# B&R Automation Studio project TD52 (part 28)

#### Ctr_CCCyclic.st
```iecst
(*******************************************************************************
Ctr_CC

This code is confidential and proprietary to the INNIO Company.
It may not be used in any form, or reproduced in any manner,
without the express written permission of the INNIO Company.
Copyright, INNIO Company, 2022

Customized modifications: -
------------------------

History:
-------
V4.x.x		14.01.2015	Walid Mari  	copied from Ctr_ECW
V4.00.1		25.06.2015	lettenbichler	twice declared par.removed
V4.11.0		28.01.2022	Perktold		included plant controller upgrade

Instructions for use:
--------------------

Outstandings:
------------
(*******************************************************************************)

PROGRAM _CYCLIC

	(* Parameter *)
	Para.tCtr_CC.W_set;
	Para.tCtr_CC.W_set2;
	Para.tCtr_CC.W_min;
	Para.tCtr_CC.W_max;
	Para.tCtr_CC.dW_up;
	Para.tCtr_CC.dW_down;
	Para.tCtr_CC.deadband;
	Para.tCtr_CC.Y_min;
	Para.tCtr_CC.Y_max;
	Para.tCtr_CC.dY_max;
	Para.tCtr_CC.Y_block;
	Para.tCtr_CC.invert;
	Para.tCtr_CC.Kp;
	Para.tCtr_CC.Tn;
	Para.tCtr_CC.Tv;
	Para.tCtr_CC.Kp_GainScheduling;
	Para.tCtr_CC.Tn_GainScheduling;
	Para.tCtr_CC.Tv_GainScheduling;

	(* Input variables *)
	tCtr_CC_In	 				:= VIS2MM.tCtr_CC_In;			(* from vis *)

	(* Input from module *)
	tCtr_CC_In.enable			:= OUT_AG.tBbBlower.Do		AND
								   Para.bCtr_CC 			AND
								   Para.bPr_CC_MS_Exist		AND
								   IN_AG.tPB2MM.bParaSetupOk;

	tCtr_CC_In.W_ext_Active		:= tCtr_CC_In.W_ext_Active;		(* from vis *)
	tCtr_CC_In.W_ext			:= 0.0;
	tCtr_CC_In.Y_set_Active		:= FALSE;
	tCtr_CC_In.Y_set			:= 0.0;
	tCtr_CC_In.X				:= IN_AG.tPr_CC.Ai;
	tCtr_CC_In.A				:= 0;
	tCtr_CC_In.W_set2_Active	:= FALSE;	(*Input to define which internal setpoint will be used TRUE = use the 2nd set point | FALSE use the normal "1st" one*)
	tCtr_CC_In.GainScheduling	:= 0.0;		(*Input for Gain Scheduling: 0.0 = use 100% of the Standard PID-Parameters | 1.0 = use 100% of the GainSched. PID Parameters | linear interpolation in between*)
	tCtr_CC_In.Y_min_cust		:= -1.0;	(*"customized" Y-Min at the current moment (The existing Y-Min parameter is the global minimum. To have an effect Y_min_cust needs to be > the parameter | -1.0 = function not used*)
	tCtr_CC_In.Y_max_cust		:= 1.0;		(*"customized" Y-Max at the current moment (The existing Y-Max parameter is the global maximum. To have an effect Y_max_cust needs to be < the parameter | 1.0 = function not used*)
	tCtr_CC_In.Retrigger		:= FALSE;	(*a rising edge on this input signals the controller to retrigger - set W on X and force the Integrator to the current Y*)

	(* Input from Visualization via OPC *)
	tCtr_CC_In.Y_man_Active;
	tCtr_CC_In.Y_man;
	tCtr_CC_In.X_min;
	tCtr_CC_In.X_max;
	tCtr_CC_In.Tune_quality;
	tCtr_CC_In.Tune_PI;
	tCtr_CC_In.Tune_PID;
	tCtr_CC_In.Tune_start;
	tCtr_CC_In.Tune_stop;
	tCtr_CC_In.Tune_takeover;

	xCtr_CC();

	(* Output variables function block *)
	(* Output to module(s) *)
	rPc_BbBlower 				:= tCtr_CC_Out.Y;	(* analog out *)

	(* Output to Visualization via OPC *)
	MM2VIS.tCtr_CC_Out			:= tCtr_CC_Out;
	VIS2MM.tCtr_CC_In			:= tCtr_CC_In;		(* write back to IN_struct for reset: Tune_takeover, X-display, ...!*)

	tCtr_CC_Out.Active;
	tCtr_CC_Out.Y;
	tCtr_CC_Out.W;
	tCtr_CC_Out.e;
	tCtr_CC_Out.Kp_tune;
	tCtr_CC_Out.Tn_tune;
	tCtr_CC_Out.Tv_tune;
	tCtr_CC_Out.status;

END_PROGRAM
```

#### Ctr_CCInit.st
```iecst
PROGRAM _INIT

	xCtr_CC.pParameter 	:= ADR(Para.tCtr_CC);
	xCtr_CC.pInput 	 	:= ADR(tCtr_CC_In);
	xCtr_CC.pOutput	 	:= ADR(tCtr_CC_Out);

	tCtr_CC_In.AlwaysUseYRamp		:= TRUE;	(*If TRUE the Y signal will always limit the change rate via the according parameter | if FALSE the Y signal will jump in case the controller is disabled (blocked or set)*)
	tCtr_CC_In.KeepYManAtBlock		:= TRUE;	(*If TRUE the controller will keep the Y-man value constant in case the controller is disabled (blocked or set) | If FALSE the blocked or set value will override the Y-man value*)
	tCtr_CC_In.Y_min_cust			:= -1.0;	(*"customized" Y-Min at the current moment (The existing Y-Min parameter is the global minimum. To have an effect Y_min_cust needs to be > the parameter | -1.0 = function not used*)
	tCtr_CC_In.Y_max_cust			:=  1.0;	(*"customized" Y-Max at the current moment (The existing Y-Max parameter is the global maximum. To have an effect Y_max_cust needs to be < the parameter | 1.0 = function not used*)
	tCtr_CC_In.StepperMode			:= FALSE;	(* TRUE = use PWM-Mode (standard mode until 4.10) | FALSE = use continuous servo drive *)
END_PROGRAM
```

### Program Logical/AuxiliariesGeneral/Ctr_ECW (IEC, version 4.12.0) - controller engine cooling water

#### Ctr_ECWCyclic.st
```iecst
(*******************************************************************************
Ctr_ECW		controller engine cooling water temperature

This code is confidential and proprietary to the INNIO Company.
It may not be used in any form, or reproduced in any manner,
without the express written permission of the INNIO Company.
Copyright, INNIO Company, 2022

Customized modifications: -
------------------------

History:
-------
V3.90.0		01.10.2012	lettenb.	new for series 9
			23.11.2012	lettenb.	write back to IN_struct added (zengerer)
V4.00.0		15.12.2014				work around(920 stapelfeld)
V4.03.0     11.01.2016              temporarily para set after controller start added
V4.03.1		03.10.2016  Fahringer	modified controller and ramp start(GeACtr with AntiWindUp)
									canceled 3 min. Tv after controller start
V4.04.0		23.03.2017	lettenb.	init restored for GeACtr with AntiWindUp
V4.05.0 	20.09.2017	Messner		Active Cooling Program added
V4.07.0		04.04.2019	Fahringer	restart the controller to initiate the setpoint ramp
			20.05.2019	Schmid		bCtrDisable was missing in tCtr_ECW_In.enable
V4.11.0		28.01.2022	Perktold	included plant controller upgrade
V4.12.0		14.12.2022	Perktold	retrigger caused by X >= WMin just once per controller activation

Instructions for use:
--------------------

Outstandings:
------------
(*******************************************************************************)

PROGRAM _CYCLIC

	(* Parameter *)
	Para.tCtr_ECW.W_set;
	Para.tCtr_ECW.W_set2;
	Para.tCtr_ECW.W_min;
	Para.tCtr_ECW.W_max;
	Para.tCtr_ECW.dW_up;
	Para.tCtr_ECW.dW_down;
	Para.tCtr_ECW.deadband;
	Para.tCtr_ECW.Y_min;
	Para.tCtr_ECW.Y_max;
	Para.tCtr_ECW.dY_max;
	Para.tCtr_ECW.Y_block;
	Para.tCtr_ECW.invert;
	Para.tCtr_ECW.Kp;
	Para.tCtr_ECW.Tn;
	Para.tCtr_ECW.Tv;
	Para.tCtr_ECW.Kp_GainScheduling;
	Para.tCtr_ECW.Tn_GainScheduling;
	Para.tCtr_ECW.Tv_GainScheduling;
	Para.tCtr_ECW.t_min_pulse_down;
	Para.tCtr_ECW.t_min_pulse_up;
	Para.tCtr_ECW.t_period_down;
	Para.tCtr_ECW.t_period_up;

	(* Input variables *)
	tCtr_ECW_In	 				:= VIS2MM.tCtr_ECW_In;			(* from vis *)

	(* Input from module *)
	tCtr_ECW_In.enable			:=	IN_AG.tPB2MM.bParaSetupOk
								AND	Para.bCtr_ECW
								AND IN_AG.bEng_Aux_Dem_CDR
								AND bCtr_ECW_Activation;

	(* start controller when actual value X reached the minimum setpoint W_min *)
	IF tCtr_ECW_In.X >= Para.tCtr_ECW.W_min THEN
		bCtr_ECW_Activation := TRUE;
	ELSE
		bCtr_ECW_Activation := tCtr_ECW_In.enable;
	END_IF;

	(* Active Cooling Program - valve setpoint *)
	IF IN_AG.bEng_Aux_Dem_CDR THEN
		tCtr_ECW_In.Y_set_Active	:= FALSE;
		tCtr_ECW_In.Y_set			:= 0.0;
	ELSE
		tCtr_ECW_In.Y_set_Active	:= bACP_Start AND NOT bACP_ECW_Cmp AND OUT_AG.tECWP1Dem.Do;
		tCtr_ECW_In.Y_set			:= 1.0;
	END_IF;

	tCtr_ECW_In.W_ext_Active	:= tCtr_ECW_In.W_ext_Active;	(* from vis *)
	tCtr_ECW_In.W_ext			:= 0.0;
	tCtr_ECW_In.X				:= IN_AG.tT_ECW.Ai;
	tCtr_ECW_In.A				:= 0;
	tCtr_ECW_In.W_set2_Active	:= FALSE;	(*Input to define which internal setpoint will be used TRUE = use the 2nd set point | FALSE use the normal "1st" one*)
	tCtr_ECW_In.GainScheduling	:= 0.0;		(*Input for Gain Scheduling: 0.0 = use 100% of the Standard PID-Parameters | 1.0 = use 100% of the GainSched. PID Parameters | linear interpolation in between*)
	tCtr_ECW_In.Y_min_cust		:= -1.0;	(*"customized" Y-Min at the current moment (The existing Y-Min parameter is the global minimum. To have an effect Y_min_cust needs to be > the parameter | -1.0 = function not used*)
	tCtr_ECW_In.Y_max_cust		:= 1.0;		(*"customized" Y-Max at the current moment (The existing Y-Max parameter is the global maximum. To have an effect Y_max_cust needs to be < the parameter | 1.0 = function not used*)

	(* retrigger controller when Ctrl.X reached the minimum set point W_min and GCB is closed  OR closure of GCB*)
	tCtr_ECW_In.Retrigger	:= (EDGEPOS(tCtr_ECW_In.X >= Para.tCtr_ECW.W_min) AND NOT bBlockRetrigger) OR EDGEPOS(IN_AG.tGCB_On.Di);

	(* block retrigger caused be X >= WMin after one execution until controller is disabled again *)
	IF tCtr_ECW_In.Retrigger AND EDGEPOS(tCtr_ECW_In.X >= Para.tCtr_ECW.W_min) THEN
		bBlockRetrigger	:= TRUE;
	ELSIF bBlockRetrigger AND NOT tCtr_ECW_In.enable THEN
		bBlockRetrigger	:= FALSE;
	END_IF;

	(* Input from Visualization via OPC *)
	tCtr_ECW_In.Y_man_Active;
	tCtr_ECW_In.Y_man;
	tCtr_ECW_In.X_min;
	tCtr_ECW_In.X_max;
	tCtr_ECW_In.Tune_quality;
	tCtr_ECW_In.Tune_PI;
	tCtr_ECW_In.Tune_PID;
	tCtr_ECW_In.Tune_start;
	tCtr_ECW_In.Tune_stop;
	tCtr_ECW_In.Tune_takeover;

	xCtr_ECW();

	(* Output variables function block *)
	(* Output to module(s) *)
	OUT_AG.tCtr_ECW_Set.Ao 	:= tCtr_ECW_Out.Y;	(* analog out *)

	(* Output to Visualization via OPC *)
	MM2VIS.tCtr_ECW_Out		:= tCtr_ECW_Out;
	VIS2MM.tCtr_ECW_In		:= tCtr_ECW_In;		(* write back to IN_struct for reset: Tune_takeover, X-display, ...!*)

	tCtr_ECW_Out.Active;
	tCtr_ECW_Out.Y;
	tCtr_ECW_Out.W;
	tCtr_ECW_Out.e;
	tCtr_ECW_Out.Kp_tune;
	tCtr_ECW_Out.Tn_tune;
	tCtr_ECW_Out.Tv_tune;
	tCtr_ECW_Out.status;

END_PROGRAM
```

#### Ctr_ECWInit.st
```iecst
PROGRAM _INIT

	xCtr_ECW.pParameter  := ADR(Para.tCtr_ECW);
	xCtr_ECW.pInput 	 := ADR(tCtr_ECW_In);
	xCtr_ECW.pOutput	 := ADR(tCtr_ECW_Out);

	tCtr_ECW_In.AlwaysUseYRamp		:= TRUE;	(*If TRUE the Y signal will always limit the change rate via the according parameter | if FALSE the Y signal will jump in case the controller is disabled (blocked or set)*)
	tCtr_ECW_In.KeepYManAtBlock		:= TRUE;	(*If TRUE the controller will keep the Y-man value constant in case the controller is disabled (blocked or set) | If FALSE the blocked or set value will override the Y-man value*)
	tCtr_ECW_In.Y_min_cust			:= -1.0;	(*"customized" Y-Min at the current moment (The existing Y-Min parameter is the global minimum. To have an effect Y_min_cust needs to be > the parameter | -1.0 = function not used*)
	tCtr_ECW_In.Y_max_cust			:=  1.0;	(*"customized" Y-Max at the current moment (The existing Y-Max parameter is the global maximum. To have an effect Y_max_cust needs to be < the parameter | 1.0 = function not used*)
	tCtr_ECW_In.StepperMode			:= FALSE;	(* TRUE = use PWM-Mode (standard mode until 4.10) | FALSE = use continuous servo drive *)

END_PROGRAM
```

#### Ctr_ECW.var
```iecst
VAR
	bCtr_ECW_Activation : BOOL; (*activation of CW controller if X is above W_min *)
	bBlockRetrigger : BOOL; (*block retrigger events*)
END_VAR
```

### Program Logical/AuxiliariesGeneral/Ctr_EOVal (IEC, version 4.12.0) - controller engine oil temperature

#### Ctr_EOValCyclic.st
```iecst
(*******************************************************************************
Ctr_EOVal		engine oil temperature control

This code is confidential and proprietary to the INNIO Company.
It may not be used in any form, or reproduced in any manner,
without the express written permission of the INNIO Company.
Copyright, INNIO Company, 2022

Customized modifications: -
------------------------

History:
-------
V3.90.0	20.03.2012	denk 		Created initial structured text code
V3.99.0	04.04.2013	lettenb.	task renamed, typ/var file removed
		03.05.2013				ctr input var's from vis added
V4.00.0	15.12.2014				work around TCV6 (920 stapelfeld)(ohne abkühlprogramm)
V4.03.0	06.07.2015				tT_EO_Mod_Out.Ai added (920 oil module, tca-redesign)
        11.01.2016              temporarily para set after controller start added
V4.03.1	08.11.2016              temporarily para set after controller start removed(GeACtr with AntiWindUp)
V4.04.0	23.03.2017	lettenb.	init restored for GeACtr with AntiWindUp
V4.05.0 20.09.2017	Messner		Active Cooling Program added
V4.11.0	28.01.2022	Perktold	included plant controller upgrade, retrigger added
V4.12.0	14.12.2022	Perktold	retrigger caused by X >= WMin just once per controller activation

Instructions for use:
--------------------

Outstandings:
------------
(*******************************************************************************)

PROGRAM _CYCLIC

	(* Parameter Oil valve controller *)
	Para.tCtr_EOVal.W_set;
	Para.tCtr_EOVal.W_set2;
	Para.tCtr_EOVal.W_min;
	Para.tCtr_EOVal.W_max;
	Para.tCtr_EOVal.dW_up;
	Para.tCtr_EOVal.dW_down;
	Para.tCtr_EOVal.deadband;
	Para.tCtr_EOVal.Y_min;
	Para.tCtr_EOVal.Y_max;
	Para.tCtr_EOVal.dY_max;
	Para.tCtr_EOVal.Y_block;
	Para.tCtr_EOVal.invert;
	Para.tCtr_EOVal.Kp;
	Para.tCtr_EOVal.Tn;
	Para.tCtr_EOVal.Tv;
	Para.tCtr_EOVal.Kp_GainScheduling;
	Para.tCtr_EOVal.Tn_GainScheduling;
	Para.tCtr_EOVal.Tv_GainScheduling;
	Para.tCtr_EOVal.t_min_pulse_down;
	Para.tCtr_EOVal.t_min_pulse_up;
	Para.tCtr_EOVal.t_period_down;
	Para.tCtr_EOVal.t_period_up;

	(* Input variables *)
	tCtr_EOVal_In	 			:= VIS2MM.tCtr_EOVal_In;			(* from Vis *)

	(* Input from module *)
	tCtr_EOVal_In.enable		:=  IN_AG.tPB2MM.bParaSetupOk
								AND Para.bCtr_EOVal_Active
								AND(IN_AG.bEng_Aux_Dem_CDR OR M_DREHZ OR bTC_CoolDownRun)
								AND bCtr_EOVal_Activation;

	(* start controller when actual value X reached the minimum setpoint W_min *)
	IF tCtr_EOVal_In.X >= Para.tCtr_EOVal.W_min THEN
		bCtr_EOVal_Activation := TRUE;
	ELSE
		bCtr_EOVal_Activation := tCtr_EOVal_In.enable;
	END_IF;

	(* Active Cooling Program - valve setpoint *)
	IF IN_AG.bEng_Aux_Dem_CDR THEN
		tCtr_EOVal_In.Y_set_Active	:= FALSE;
		tCtr_EOVal_In.Y_set			:= 0.0;
	ELSE
		tCtr_EOVal_In.Y_set_Active	:= bACP_Start AND NOT bACP_EO_Cmp AND OUT_AG.tEOP1AC_Dem.Do;
		tCtr_EOVal_In.Y_set			:= 1.0;
	END_IF;

	tCtr_EOVal_In.W_ext_Active	:= tCtr_EOVal_In.W_ext_Active;
	tCtr_EOVal_In.W_ext			:= 0.0;
//	IF IN_AG.tT_EO_Mod_Out.GoodQual THEN tCtr_EOVal_In.X := IN_AG.tT_EO_Mod_Out.Ai; (* oil module *)
//	ELSE                                 tCtr_EOVal_In.X := IN_AG.tT_EO.Ai;         (* engine *)
//	END_IF;
	tCtr_EOVal_In.X 			:= IN_AG.tT_EO.Ai;
	tCtr_EOVal_In.A				:= 0.0;
	tCtr_EOVal_In.W_set2_Active	:= FALSE;	(*Input to define which internal setpoint will be used TRUE = use the 2nd set point | FALSE use the normal "1st" one*)
	tCtr_EOVal_In.GainScheduling:= 0.0;		(*Input for Gain Scheduling: 0.0 = use 100% of the Standard PID-Parameters | 1.0 = use 100% of the GainSched. PID Parameters | linear interpolation in between*)
	tCtr_EOVal_In.Y_min_cust	:= -1.0;	(*"customized" Y-Min at the current moment (The existing Y-Min parameter is the global minimum. To have an effect Y_min_cust needs to be > the parameter | -1.0 = function not used*)
	tCtr_EOVal_In.Y_max_cust	:= 1.0;		(*"customized" Y-Max at the current moment (The existing Y-Max parameter is the global maximum. To have an effect Y_max_cust needs to be < the parameter | 1.0 = function not used*)

	(* retrigger controller when Ctrl.X reached the minimum set point W_min OR closure of GCB*)
	tCtr_EOVal_In.Retrigger		:= (EDGEPOS(tCtr_EOVal_In.X >= Para.tCtr_EOVal.W_min) AND NOT bBlockRetrigger) OR EDGEPOS(IN_AG.tGCB_On.Di);

	(* block retrigger caused be X >= WMin after one execution until controller is disabled again *)
	IF tCtr_EOVal_In.Retrigger AND EDGEPOS(tCtr_EOVal_In.X >= Para.tCtr_EOVal.W_min) THEN
		bBlockRetrigger	:= TRUE;
	ELSIF bBlockRetrigger AND NOT tCtr_EOVal_In.enable THEN
		bBlockRetrigger	:= FALSE;
	END_IF;

	(* Input from Visualization via OPC *)
	tCtr_EOVal_In.Y_man_Active;
	tCtr_EOVal_In.Y_man;
	tCtr_EOVal_In.X_min;
	tCtr_EOVal_In.X_max;
	tCtr_EOVal_In.Tune_quality;
	tCtr_EOVal_In.Tune_PI;
	tCtr_EOVal_In.Tune_PID;
	tCtr_EOVal_In.Tune_start;
	tCtr_EOVal_In.Tune_stop;
	tCtr_EOVal_In.Tune_takeover;

	xCtr_EOVal();

	(* Output variables  Oil valve controller function block *)
	(* Output to module(s) *)
	OUT_AG.tOV_Ctrl_Set.Ao 		:= tCtr_EOVal_Out.Y;	(* analog out *)

	(* Output to Visualization via OPC *)
	MM2VIS.tCtr_EOVal_Out		:= tCtr_EOVal_Out;
	VIS2MM.tCtr_EOVal_In		:= tCtr_EOVal_In;		(* write back to IN_struct for reset: Tune_takeover, X-display, ...!*)

	tCtr_EOVal_Out.Active;
	tCtr_EOVal_Out.Y;
	tCtr_EOVal_Out.W;
	tCtr_EOVal_Out.e;
	tCtr_EOVal_Out.Kp_tune;
	tCtr_EOVal_Out.Tn_tune;
	tCtr_EOVal_Out.Tv_tune;
	tCtr_EOVal_Out.status;

END_PROGRAM
```

#### Ctr_EOValInit.st
```iecst
PROGRAM _INIT

	xCtr_EOVal.pParameter 	:= ADR(Para.tCtr_EOVal);
	xCtr_EOVal.pInput 		:= ADR(tCtr_EOVal_In);
	xCtr_EOVal.pOutput	 	:= ADR(tCtr_EOVal_Out);

	tCtr_EOVal_In.AlwaysUseYRamp		:= TRUE;	(*If TRUE the Y signal will always limit the change rate via the according parameter | if FALSE the Y signal will jump in case the controller is disabled (blocked or set)*)
	tCtr_EOVal_In.KeepYManAtBlock		:= TRUE;	(*If TRUE the controller will keep the Y-man value constant in case the controller is disabled (blocked or set) | If FALSE the blocked or set value will override the Y-man value*)
	tCtr_EOVal_In.Y_min_cust			:= -1.0;	(*"customized" Y-Min at the current moment (The existing Y-Min parameter is the global minimum. To have an effect Y_min_cust needs to be > the parameter | -1.0 = function not used*)
	tCtr_EOVal_In.Y_max_cust			:=  1.0;	(*"customized" Y-Max at the current moment (The existing Y-Max parameter is the global maximum. To have an effect Y_max_cust needs to be < the parameter | 1.0 = function not used*)
	tCtr_EOVal_In.StepperMode			:= FALSE;	(* TRUE = use PWM-Mode (standard mode until 4.10) | FALSE = use continuous servo drive *)

END_PROGRAM
```

#### Ctr_EOVal.var
```iecst
VAR
	bCtr_EOVal_Activation : BOOL; (*activation of CW controller if X is above W_min *)
	bBlockRetrigger : BOOL; (*block retrigger events*)
END_VAR

VAR CONSTANT

END_VAR
```

### Program Logical/AuxiliariesGeneral/Ctr_EOVal_LT (IEC, version 4.11.0) - controller engine oil temperature LT circuit

#### Ctr_EOVal_LTCyclic.st
```iecst
(*******************************************************************************
Ctr_EOVal_LT		engine oil temperature control LT circuit

This code is confidential AND proprietary to the INNIO Company.
It may NOT be used in any form, or reproduced in any manner,
without the express written permission of the INNIO Company.
Copyright, INNIO Company, 2022

Customized modifications: -
------------------------

History:
-------
V3.90.0	20.03.2012	denk 		Created initial structured text code
V3.99.0	04.04.2013	lettenb.	task renamed, typ/var file removed
		03.05.2013				ctr input var's from vis added
V4.00.0	15.12.2014				work around TCV1 (920 stapelfeld)(ohne abkühlprogramm)
V4.03.0	06.07.2015				tT_EO_Mod_Out.Ai added (920 ECW-modul)
		14.03.2016				tCtr_EOVal_In.X -> tCtr_EOVal_LT_In.X, bugfix
V4.04.0	23.03.2017	lettenb.	tCtr_EOVal_LT_In.X according Ctr_EOVal
V4.11.0	28.01.2022	Perktold	included plant controller upgrade

(*******************************************************************************)

PROGRAM _CYCLIC

	(* Parameter Oil valve controller *)
	Para.tCtr_EOVal_LT.W_set;
	Para.tCtr_EOVal_LT.W_set2;
	Para.tCtr_EOVal_LT.W_min;
	Para.tCtr_EOVal_LT.W_max;
	Para.tCtr_EOVal_LT.dW_up;
	Para.tCtr_EOVal_LT.dW_down;
	Para.tCtr_EOVal_LT.deadband;
	Para.tCtr_EOVal_LT.Y_min;
	Para.tCtr_EOVal_LT.Y_max;
	Para.tCtr_EOVal_LT.dY_max;
	Para.tCtr_EOVal_LT.Y_block;
	Para.tCtr_EOVal_LT.invert;
	Para.tCtr_EOVal_LT.Kp;
	Para.tCtr_EOVal_LT.Tn;
	Para.tCtr_EOVal_LT.Tv;
	Para.tCtr_EOVal_LT.Kp_GainScheduling;
	Para.tCtr_EOVal_LT.Tn_GainScheduling;
	Para.tCtr_EOVal_LT.Tv_GainScheduling;
	Para.tCtr_EOVal_LT.t_min_pulse_down;
	Para.tCtr_EOVal_LT.t_min_pulse_up;
	Para.tCtr_EOVal_LT.t_period_down;
	Para.tCtr_EOVal_LT.t_period_up;

	(* Input variables *)
	tCtr_EOVal_LT_In	 			:= VIS2MM.tCtr_EOVal_LT_In;			(* from Vis *)

	(* Input from module *)
	tCtr_EOVal_LT_In.enable		:=  IN_AG.tPB2MM.bParaSetupOk
								AND Para.bCtr_EOVal_LT_Active
								AND(IN_AG.bEng_Aux_Dem_CDR OR bPreLubeDem OR bTC_CoolDownRun);
	tCtr_EOVal_LT_In.W_ext_Active	:= tCtr_EOVal_LT_In.W_ext_Active;
	tCtr_EOVal_LT_In.W_ext			:= 50.0;
	tCtr_EOVal_LT_In.Y_set_Active	:= OUT_AG.bMsg2102;
	tCtr_EOVal_LT_In.Y_set 			:= 0.5;
//	IF IN_AG.tT_EO_Mod_Out.GoodQual THEN tCtr_EOVal_LT_In.X := IN_AG.tT_EO_Mod_Out.Ai; (* 920 ECW-module *)
//	ELSE                                 tCtr_EOVal_LT_In.X := IN_AG.tT_EO.Ai;
//	END_IF;
	tCtr_EOVal_LT_In.X 				:= IN_AG.tT_EO.Ai;
	tCtr_EOVal_LT_In.A				:= 0.0;
	tCtr_EOVal_LT_In.W_set2_Active	:= FALSE;	(*Input to define which internal setpoint will be used TRUE = use the 2nd set point | FALSE use the normal "1st" one*)
	tCtr_EOVal_LT_In.GainScheduling	:= 0.0;		(*Input for Gain Scheduling: 0.0 = use 100% of the Standard PID-Parameters | 1.0 = use 100% of the GainSched. PID Parameters | linear interpolation in between*)
	tCtr_EOVal_LT_In.Y_min_cust		:= -1.0;	(*"customized" Y-Min at the current moment (The existing Y-Min parameter is the global minimum. To have an effect Y_min_cust needs to be > the parameter | -1.0 = function not used*)
	tCtr_EOVal_LT_In.Y_max_cust		:= 1.0;		(*"customized" Y-Max at the current moment (The existing Y-Max parameter is the global maximum. To have an effect Y_max_cust needs to be < the parameter | 1.0 = function not used*)
	tCtr_EOVal_LT_In.Retrigger		:= FALSE;	(*a rising edge on this input signals the controller to retrigger - set W on X and force the Integrator to the current Y*)

	(* Input from Visualization via OPC *)
	tCtr_EOVal_LT_In.Y_man_Active;
	tCtr_EOVal_LT_In.Y_man;
	tCtr_EOVal_LT_In.X_min;
	tCtr_EOVal_LT_In.X_max;
	tCtr_EOVal_LT_In.Tune_quality;
	tCtr_EOVal_LT_In.Tune_PI;
	tCtr_EOVal_LT_In.Tune_PID;
	tCtr_EOVal_LT_In.Tune_start;
	tCtr_EOVal_LT_In.Tune_stop;
	tCtr_EOVal_LT_In.Tune_takeover;

	xCtr_EOVal_LT();

	(* Output variables  Oil valve controller function block *)
	(* Output to module(s) *)
	OUT_AG.tEOVal_LT_Set.Ao 	:= tCtr_EOVal_LT_Out.Y;	(* analog out *)

	(* Output to Visualization via OPC *)
	MM2VIS.tCtr_EOVal_LT_Out	:= tCtr_EOVal_LT_Out;
	VIS2MM.tCtr_EOVal_LT_In		:= tCtr_EOVal_LT_In;		(* write back to IN_struct for reset: Tune_takeover, X-display, ...!*)

	tCtr_EOVal_LT_Out.Active;
	tCtr_EOVal_LT_Out.Y;
	tCtr_EOVal_LT_Out.W;
	tCtr_EOVal_LT_Out.e;
	tCtr_EOVal_LT_Out.Kp_tune;
	tCtr_EOVal_LT_Out.Tn_tune;
	tCtr_EOVal_LT_Out.Tv_tune;
	tCtr_EOVal_LT_Out.status;

END_PROGRAM
```

#### Ctr_EOVal_LTInit.st
```iecst
PROGRAM _INIT

	xCtr_EOVal_LT.pParameter 	:= ADR(Para.tCtr_EOVal_LT);
	xCtr_EOVal_LT.pInput 		:= ADR(tCtr_EOVal_LT_In);
	xCtr_EOVal_LT.pOutput	 	:= ADR(tCtr_EOVal_LT_Out);

	tCtr_EOVal_LT_In.AlwaysUseYRamp		:= TRUE;	(*If TRUE the Y signal will always limit the change rate via the according parameter | if FALSE the Y signal will jump in case the controller is disabled (blocked or set)*)
	tCtr_EOVal_LT_In.KeepYManAtBlock	:= TRUE;	(*If TRUE the controller will keep the Y-man value constant in case the controller is disabled (blocked or set) | If FALSE the blocked or set value will override the Y-man value*)
	tCtr_EOVal_LT_In.Y_min_cust			:= -1.0;	(*"customized" Y-Min at the current moment (The existing Y-Min parameter is the global minimum. To have an effect Y_min_cust needs to be > the parameter | -1.0 = function not used*)
	tCtr_EOVal_LT_In.Y_max_cust			:=  1.0;	(*"customized" Y-Max at the current moment (The existing Y-Max parameter is the global maximum. To have an effect Y_max_cust needs to be < the parameter | 1.0 = function not used*)
	tCtr_EOVal_LT_In.StepperMode		:= FALSE;	(* TRUE = use PWM-Mode (standard mode until 4.10) | FALSE = use continuous servo drive *)

END_PROGRAM
```

### Program Logical/AuxiliariesGeneral/MsgAG (IEC) - messages
